// TIA Portal V20 export
FUNCTION_BLOCK "FB_What_Was_Read"   // FB7, LAD
{ S7_Optimized_Access := 'TRUE' }
// stored: AutoNumber false, MemoryReserve 100, SetENOAutomatically false
   VAR_INPUT
      Read_Data_In : "SR-X100W_Read_Data";
   END_VAR
   VAR_OUTPUT
      Read_Data_Out : String[136];
      Serial_Number : String[17];
   END_VAR
BEGIN

REGION Network 1
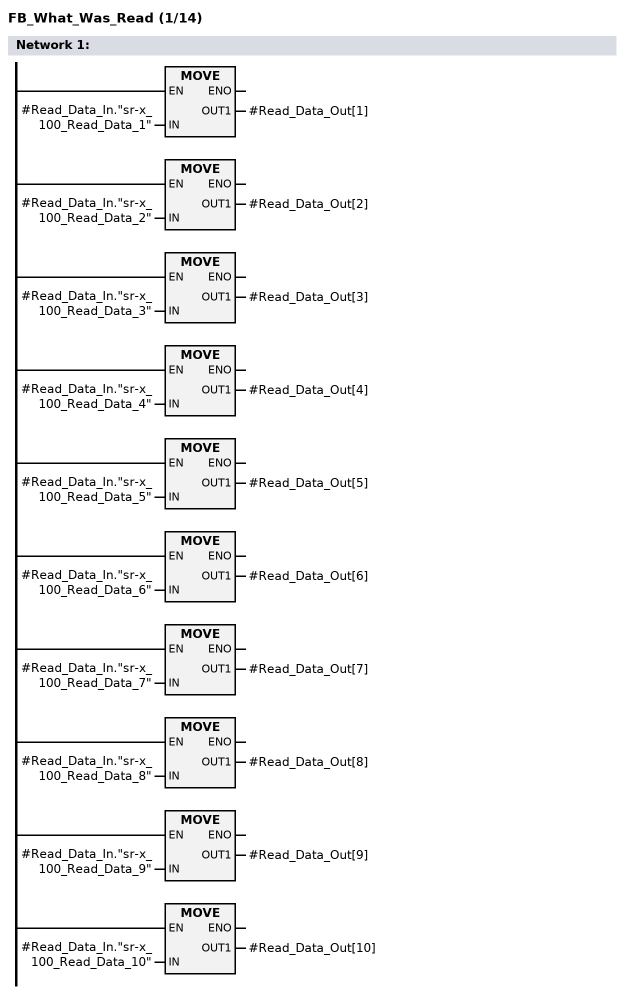
   RUNG wire#powerrail
      Move(in := #Read_Data_In."sr-x_100_Read_Data_1", out1 => #Read_Data_Out[1])
   END_RUNG
   RUNG wire#powerrail
      Move(in := #Read_Data_In."sr-x_100_Read_Data_2", out1 => #Read_Data_Out[2])
   END_RUNG
   RUNG wire#powerrail
      Move(in := #Read_Data_In."sr-x_100_Read_Data_3", out1 => #Read_Data_Out[3])
   END_RUNG
   RUNG wire#powerrail
      Move(in := #Read_Data_In."sr-x_100_Read_Data_4", out1 => #Read_Data_Out[4])
   END_RUNG
   RUNG wire#powerrail
      Move(in := #Read_Data_In."sr-x_100_Read_Data_5", out1 => #Read_Data_Out[5])
   END_RUNG
   RUNG wire#powerrail
      Move(in := #Read_Data_In."sr-x_100_Read_Data_6", out1 => #Read_Data_Out[6])
   END_RUNG
   RUNG wire#powerrail
      Move(in := #Read_Data_In."sr-x_100_Read_Data_7", out1 => #Read_Data_Out[7])
   END_RUNG
   RUNG wire#powerrail
      Move(in := #Read_Data_In."sr-x_100_Read_Data_8", out1 => #Read_Data_Out[8])
   END_RUNG
   RUNG wire#powerrail
      Move(in := #Read_Data_In."sr-x_100_Read_Data_9", out1 => #Read_Data_Out[9])
   END_RUNG
   RUNG wire#powerrail
      Move(in := #Read_Data_In."sr-x_100_Read_Data_10", out1 => #Read_Data_Out[10])
   END_RUNG
   // the same network as SCL:
   #Read_Data_Out[1] := #Read_Data_In."sr-x_100_Read_Data_1";
   #Read_Data_Out[2] := #Read_Data_In."sr-x_100_Read_Data_2";
   #Read_Data_Out[3] := #Read_Data_In."sr-x_100_Read_Data_3";
   #Read_Data_Out[4] := #Read_Data_In."sr-x_100_Read_Data_4";
   #Read_Data_Out[5] := #Read_Data_In."sr-x_100_Read_Data_5";
   #Read_Data_Out[6] := #Read_Data_In."sr-x_100_Read_Data_6";
   #Read_Data_Out[7] := #Read_Data_In."sr-x_100_Read_Data_7";
   #Read_Data_Out[8] := #Read_Data_In."sr-x_100_Read_Data_8";
   #Read_Data_Out[9] := #Read_Data_In."sr-x_100_Read_Data_9";
   #Read_Data_Out[10] := #Read_Data_In."sr-x_100_Read_Data_10";
END_REGION

REGION Network 2
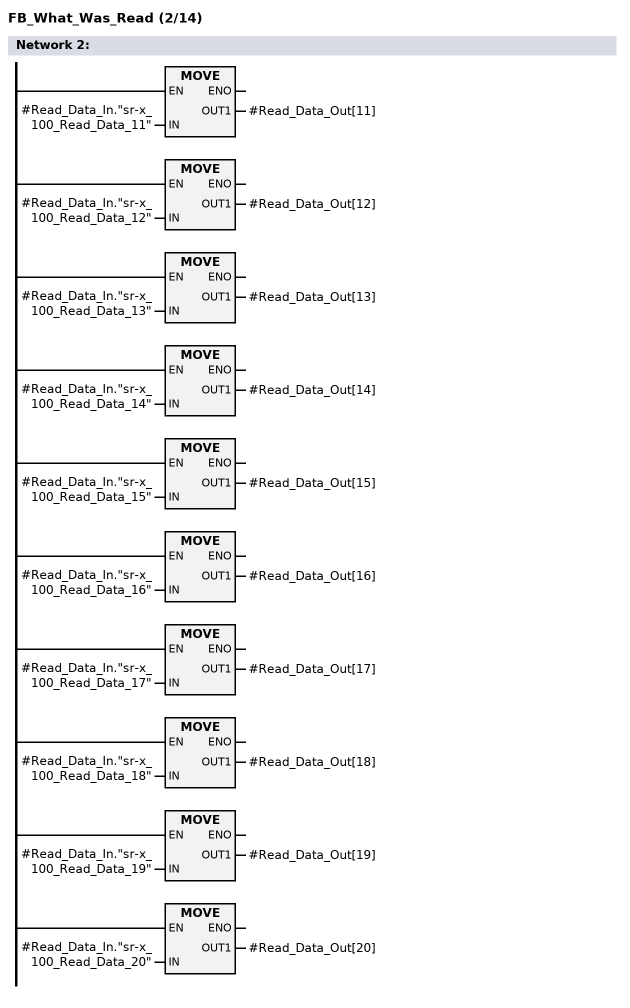
   RUNG wire#powerrail
      Move(in := #Read_Data_In."sr-x_100_Read_Data_11", out1 => #Read_Data_Out[11])
   END_RUNG
   RUNG wire#powerrail
      Move(in := #Read_Data_In."sr-x_100_Read_Data_12", out1 => #Read_Data_Out[12])
   END_RUNG
   RUNG wire#powerrail
      Move(in := #Read_Data_In."sr-x_100_Read_Data_13", out1 => #Read_Data_Out[13])
   END_RUNG
   RUNG wire#powerrail
      Move(in := #Read_Data_In."sr-x_100_Read_Data_14", out1 => #Read_Data_Out[14])
   END_RUNG
   RUNG wire#powerrail
      Move(in := #Read_Data_In."sr-x_100_Read_Data_15", out1 => #Read_Data_Out[15])
   END_RUNG
   RUNG wire#powerrail
      Move(in := #Read_Data_In."sr-x_100_Read_Data_16", out1 => #Read_Data_Out[16])
   END_RUNG
   RUNG wire#powerrail
      Move(in := #Read_Data_In."sr-x_100_Read_Data_17", out1 => #Read_Data_Out[17])
   END_RUNG
   RUNG wire#powerrail
      Move(in := #Read_Data_In."sr-x_100_Read_Data_18", out1 => #Read_Data_Out[18])
   END_RUNG
   RUNG wire#powerrail
      Move(in := #Read_Data_In."sr-x_100_Read_Data_19", out1 => #Read_Data_Out[19])
   END_RUNG
   RUNG wire#powerrail
      Move(in := #Read_Data_In."sr-x_100_Read_Data_20", out1 => #Read_Data_Out[20])
   END_RUNG
   // the same network as SCL:
   #Read_Data_Out[11] := #Read_Data_In."sr-x_100_Read_Data_11";
   #Read_Data_Out[12] := #Read_Data_In."sr-x_100_Read_Data_12";
   #Read_Data_Out[13] := #Read_Data_In."sr-x_100_Read_Data_13";
   #Read_Data_Out[14] := #Read_Data_In."sr-x_100_Read_Data_14";
   #Read_Data_Out[15] := #Read_Data_In."sr-x_100_Read_Data_15";
   #Read_Data_Out[16] := #Read_Data_In."sr-x_100_Read_Data_16";
   #Read_Data_Out[17] := #Read_Data_In."sr-x_100_Read_Data_17";
   #Read_Data_Out[18] := #Read_Data_In."sr-x_100_Read_Data_18";
   #Read_Data_Out[19] := #Read_Data_In."sr-x_100_Read_Data_19";
   #Read_Data_Out[20] := #Read_Data_In."sr-x_100_Read_Data_20";
END_REGION

REGION Network 3
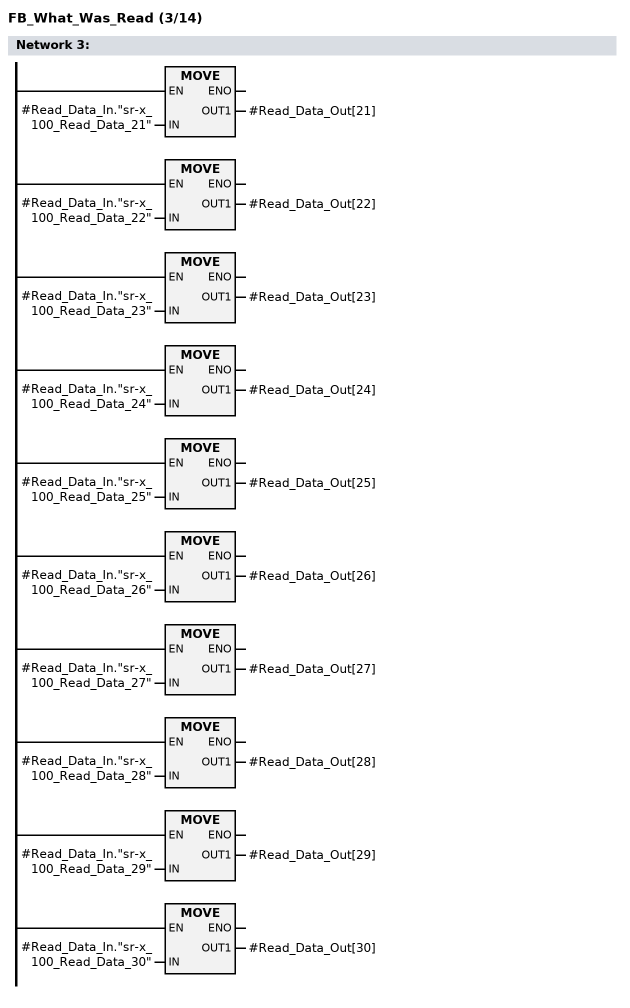
   RUNG wire#powerrail
      Move(in := #Read_Data_In."sr-x_100_Read_Data_21", out1 => #Read_Data_Out[21])
   END_RUNG
   RUNG wire#powerrail
      Move(in := #Read_Data_In."sr-x_100_Read_Data_22", out1 => #Read_Data_Out[22])
   END_RUNG
   RUNG wire#powerrail
      Move(in := #Read_Data_In."sr-x_100_Read_Data_23", out1 => #Read_Data_Out[23])
   END_RUNG
   RUNG wire#powerrail
      Move(in := #Read_Data_In."sr-x_100_Read_Data_24", out1 => #Read_Data_Out[24])
   END_RUNG
   RUNG wire#powerrail
      Move(in := #Read_Data_In."sr-x_100_Read_Data_25", out1 => #Read_Data_Out[25])
   END_RUNG
   RUNG wire#powerrail
      Move(in := #Read_Data_In."sr-x_100_Read_Data_26", out1 => #Read_Data_Out[26])
   END_RUNG
   RUNG wire#powerrail
      Move(in := #Read_Data_In."sr-x_100_Read_Data_27", out1 => #Read_Data_Out[27])
   END_RUNG
   RUNG wire#powerrail
      Move(in := #Read_Data_In."sr-x_100_Read_Data_28", out1 => #Read_Data_Out[28])
   END_RUNG
   RUNG wire#powerrail
      Move(in := #Read_Data_In."sr-x_100_Read_Data_29", out1 => #Read_Data_Out[29])
   END_RUNG
   RUNG wire#powerrail
      Move(in := #Read_Data_In."sr-x_100_Read_Data_30", out1 => #Read_Data_Out[30])
   END_RUNG
   // the same network as SCL:
   #Read_Data_Out[21] := #Read_Data_In."sr-x_100_Read_Data_21";
   #Read_Data_Out[22] := #Read_Data_In."sr-x_100_Read_Data_22";
   #Read_Data_Out[23] := #Read_Data_In."sr-x_100_Read_Data_23";
   #Read_Data_Out[24] := #Read_Data_In."sr-x_100_Read_Data_24";
   #Read_Data_Out[25] := #Read_Data_In."sr-x_100_Read_Data_25";
   #Read_Data_Out[26] := #Read_Data_In."sr-x_100_Read_Data_26";
   #Read_Data_Out[27] := #Read_Data_In."sr-x_100_Read_Data_27";
   #Read_Data_Out[28] := #Read_Data_In."sr-x_100_Read_Data_28";
   #Read_Data_Out[29] := #Read_Data_In."sr-x_100_Read_Data_29";
   #Read_Data_Out[30] := #Read_Data_In."sr-x_100_Read_Data_30";
END_REGION

REGION Network 4
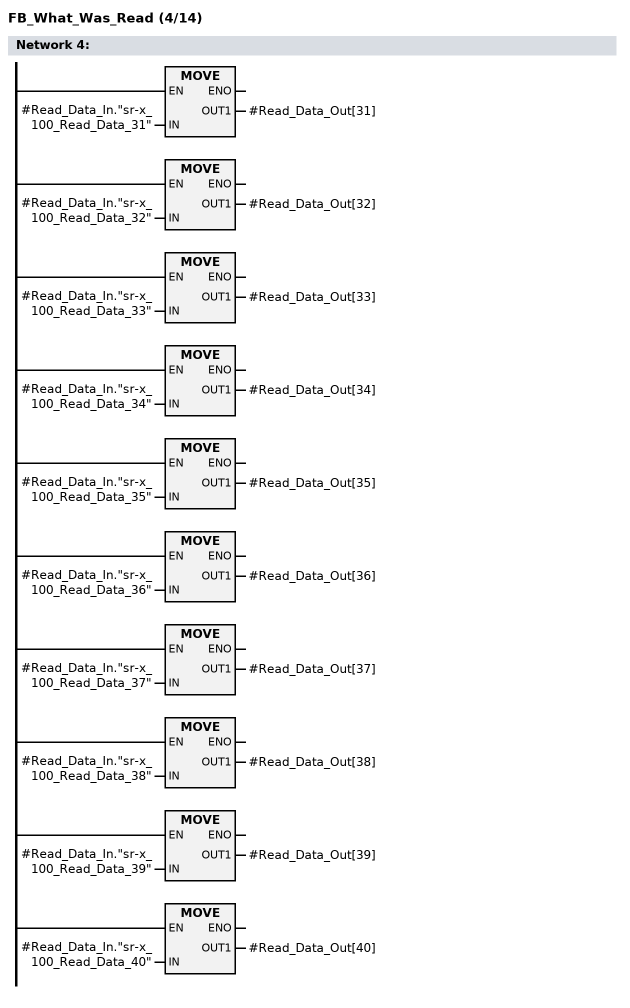
   RUNG wire#powerrail
      Move(in := #Read_Data_In."sr-x_100_Read_Data_31", out1 => #Read_Data_Out[31])
   END_RUNG
   RUNG wire#powerrail
      Move(in := #Read_Data_In."sr-x_100_Read_Data_32", out1 => #Read_Data_Out[32])
   END_RUNG
   RUNG wire#powerrail
      Move(in := #Read_Data_In."sr-x_100_Read_Data_33", out1 => #Read_Data_Out[33])
   END_RUNG
   RUNG wire#powerrail
      Move(in := #Read_Data_In."sr-x_100_Read_Data_34", out1 => #Read_Data_Out[34])
   END_RUNG
   RUNG wire#powerrail
      Move(in := #Read_Data_In."sr-x_100_Read_Data_35", out1 => #Read_Data_Out[35])
   END_RUNG
   RUNG wire#powerrail
      Move(in := #Read_Data_In."sr-x_100_Read_Data_36", out1 => #Read_Data_Out[36])
   END_RUNG
   RUNG wire#powerrail
      Move(in := #Read_Data_In."sr-x_100_Read_Data_37", out1 => #Read_Data_Out[37])
   END_RUNG
   RUNG wire#powerrail
      Move(in := #Read_Data_In."sr-x_100_Read_Data_38", out1 => #Read_Data_Out[38])
   END_RUNG
   RUNG wire#powerrail
      Move(in := #Read_Data_In."sr-x_100_Read_Data_39", out1 => #Read_Data_Out[39])
   END_RUNG
   RUNG wire#powerrail
      Move(in := #Read_Data_In."sr-x_100_Read_Data_40", out1 => #Read_Data_Out[40])
   END_RUNG
   // the same network as SCL:
   #Read_Data_Out[31] := #Read_Data_In."sr-x_100_Read_Data_31";
   #Read_Data_Out[32] := #Read_Data_In."sr-x_100_Read_Data_32";
   #Read_Data_Out[33] := #Read_Data_In."sr-x_100_Read_Data_33";
   #Read_Data_Out[34] := #Read_Data_In."sr-x_100_Read_Data_34";
   #Read_Data_Out[35] := #Read_Data_In."sr-x_100_Read_Data_35";
   #Read_Data_Out[36] := #Read_Data_In."sr-x_100_Read_Data_36";
   #Read_Data_Out[37] := #Read_Data_In."sr-x_100_Read_Data_37";
   #Read_Data_Out[38] := #Read_Data_In."sr-x_100_Read_Data_38";
   #Read_Data_Out[39] := #Read_Data_In."sr-x_100_Read_Data_39";
   #Read_Data_Out[40] := #Read_Data_In."sr-x_100_Read_Data_40";
END_REGION

REGION Network 5
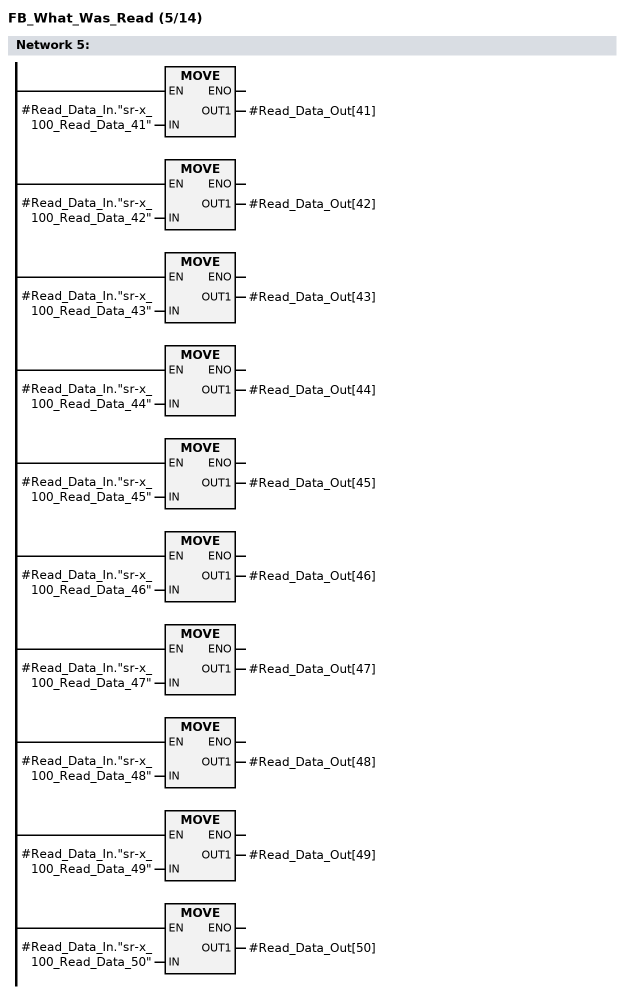
   RUNG wire#powerrail
      Move(in := #Read_Data_In."sr-x_100_Read_Data_41", out1 => #Read_Data_Out[41])
   END_RUNG
   RUNG wire#powerrail
      Move(in := #Read_Data_In."sr-x_100_Read_Data_42", out1 => #Read_Data_Out[42])
   END_RUNG
   RUNG wire#powerrail
      Move(in := #Read_Data_In."sr-x_100_Read_Data_43", out1 => #Read_Data_Out[43])
   END_RUNG
   RUNG wire#powerrail
      Move(in := #Read_Data_In."sr-x_100_Read_Data_44", out1 => #Read_Data_Out[44])
   END_RUNG
   RUNG wire#powerrail
      Move(in := #Read_Data_In."sr-x_100_Read_Data_45", out1 => #Read_Data_Out[45])
   END_RUNG
   RUNG wire#powerrail
      Move(in := #Read_Data_In."sr-x_100_Read_Data_46", out1 => #Read_Data_Out[46])
   END_RUNG
   RUNG wire#powerrail
      Move(in := #Read_Data_In."sr-x_100_Read_Data_47", out1 => #Read_Data_Out[47])
   END_RUNG
   RUNG wire#powerrail
      Move(in := #Read_Data_In."sr-x_100_Read_Data_48", out1 => #Read_Data_Out[48])
   END_RUNG
   RUNG wire#powerrail
      Move(in := #Read_Data_In."sr-x_100_Read_Data_49", out1 => #Read_Data_Out[49])
   END_RUNG
   RUNG wire#powerrail
      Move(in := #Read_Data_In."sr-x_100_Read_Data_50", out1 => #Read_Data_Out[50])
   END_RUNG
   // the same network as SCL:
   #Read_Data_Out[41] := #Read_Data_In."sr-x_100_Read_Data_41";
   #Read_Data_Out[42] := #Read_Data_In."sr-x_100_Read_Data_42";
   #Read_Data_Out[43] := #Read_Data_In."sr-x_100_Read_Data_43";
   #Read_Data_Out[44] := #Read_Data_In."sr-x_100_Read_Data_44";
   #Read_Data_Out[45] := #Read_Data_In."sr-x_100_Read_Data_45";
   #Read_Data_Out[46] := #Read_Data_In."sr-x_100_Read_Data_46";
   #Read_Data_Out[47] := #Read_Data_In."sr-x_100_Read_Data_47";
   #Read_Data_Out[48] := #Read_Data_In."sr-x_100_Read_Data_48";
   #Read_Data_Out[49] := #Read_Data_In."sr-x_100_Read_Data_49";
   #Read_Data_Out[50] := #Read_Data_In."sr-x_100_Read_Data_50";
END_REGION

REGION Network 6
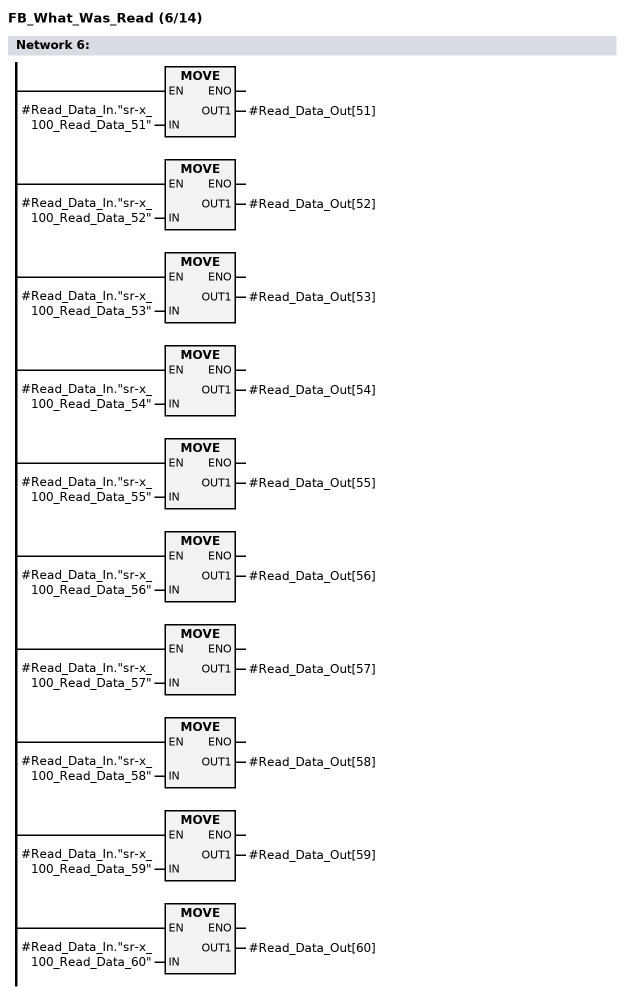
   RUNG wire#powerrail
      Move(in := #Read_Data_In."sr-x_100_Read_Data_51", out1 => #Read_Data_Out[51])
   END_RUNG
   RUNG wire#powerrail
      Move(in := #Read_Data_In."sr-x_100_Read_Data_52", out1 => #Read_Data_Out[52])
   END_RUNG
   RUNG wire#powerrail
      Move(in := #Read_Data_In."sr-x_100_Read_Data_53", out1 => #Read_Data_Out[53])
   END_RUNG
   RUNG wire#powerrail
      Move(in := #Read_Data_In."sr-x_100_Read_Data_54", out1 => #Read_Data_Out[54])
   END_RUNG
   RUNG wire#powerrail
      Move(in := #Read_Data_In."sr-x_100_Read_Data_55", out1 => #Read_Data_Out[55])
   END_RUNG
   RUNG wire#powerrail
      Move(in := #Read_Data_In."sr-x_100_Read_Data_56", out1 => #Read_Data_Out[56])
   END_RUNG
   RUNG wire#powerrail
      Move(in := #Read_Data_In."sr-x_100_Read_Data_57", out1 => #Read_Data_Out[57])
   END_RUNG
   RUNG wire#powerrail
      Move(in := #Read_Data_In."sr-x_100_Read_Data_58", out1 => #Read_Data_Out[58])
   END_RUNG
   RUNG wire#powerrail
      Move(in := #Read_Data_In."sr-x_100_Read_Data_59", out1 => #Read_Data_Out[59])
   END_RUNG
   RUNG wire#powerrail
      Move(in := #Read_Data_In."sr-x_100_Read_Data_60", out1 => #Read_Data_Out[60])
   END_RUNG
   // the same network as SCL:
   #Read_Data_Out[51] := #Read_Data_In."sr-x_100_Read_Data_51";
   #Read_Data_Out[52] := #Read_Data_In."sr-x_100_Read_Data_52";
   #Read_Data_Out[53] := #Read_Data_In."sr-x_100_Read_Data_53";
   #Read_Data_Out[54] := #Read_Data_In."sr-x_100_Read_Data_54";
   #Read_Data_Out[55] := #Read_Data_In."sr-x_100_Read_Data_55";
   #Read_Data_Out[56] := #Read_Data_In."sr-x_100_Read_Data_56";
   #Read_Data_Out[57] := #Read_Data_In."sr-x_100_Read_Data_57";
   #Read_Data_Out[58] := #Read_Data_In."sr-x_100_Read_Data_58";
   #Read_Data_Out[59] := #Read_Data_In."sr-x_100_Read_Data_59";
   #Read_Data_Out[60] := #Read_Data_In."sr-x_100_Read_Data_60";
END_REGION

REGION Network 7
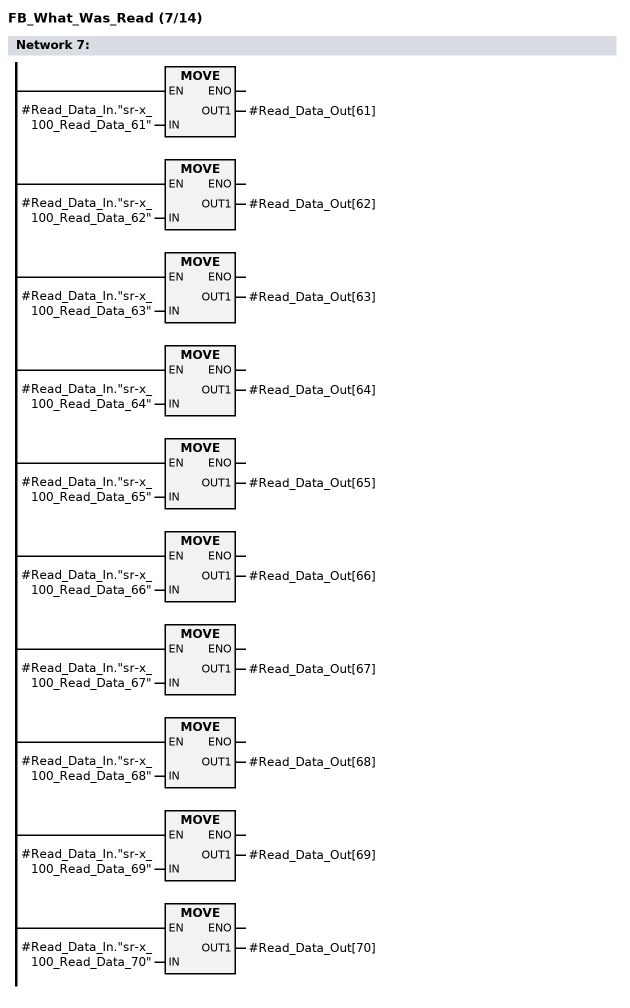
   RUNG wire#powerrail
      Move(in := #Read_Data_In."sr-x_100_Read_Data_61", out1 => #Read_Data_Out[61])
   END_RUNG
   RUNG wire#powerrail
      Move(in := #Read_Data_In."sr-x_100_Read_Data_62", out1 => #Read_Data_Out[62])
   END_RUNG
   RUNG wire#powerrail
      Move(in := #Read_Data_In."sr-x_100_Read_Data_63", out1 => #Read_Data_Out[63])
   END_RUNG
   RUNG wire#powerrail
      Move(in := #Read_Data_In."sr-x_100_Read_Data_64", out1 => #Read_Data_Out[64])
   END_RUNG
   RUNG wire#powerrail
      Move(in := #Read_Data_In."sr-x_100_Read_Data_65", out1 => #Read_Data_Out[65])
   END_RUNG
   RUNG wire#powerrail
      Move(in := #Read_Data_In."sr-x_100_Read_Data_66", out1 => #Read_Data_Out[66])
   END_RUNG
   RUNG wire#powerrail
      Move(in := #Read_Data_In."sr-x_100_Read_Data_67", out1 => #Read_Data_Out[67])
   END_RUNG
   RUNG wire#powerrail
      Move(in := #Read_Data_In."sr-x_100_Read_Data_68", out1 => #Read_Data_Out[68])
   END_RUNG
   RUNG wire#powerrail
      Move(in := #Read_Data_In."sr-x_100_Read_Data_69", out1 => #Read_Data_Out[69])
   END_RUNG
   RUNG wire#powerrail
      Move(in := #Read_Data_In."sr-x_100_Read_Data_70", out1 => #Read_Data_Out[70])
   END_RUNG
   // the same network as SCL:
   #Read_Data_Out[61] := #Read_Data_In."sr-x_100_Read_Data_61";
   #Read_Data_Out[62] := #Read_Data_In."sr-x_100_Read_Data_62";
   #Read_Data_Out[63] := #Read_Data_In."sr-x_100_Read_Data_63";
   #Read_Data_Out[64] := #Read_Data_In."sr-x_100_Read_Data_64";
   #Read_Data_Out[65] := #Read_Data_In."sr-x_100_Read_Data_65";
   #Read_Data_Out[66] := #Read_Data_In."sr-x_100_Read_Data_66";
   #Read_Data_Out[67] := #Read_Data_In."sr-x_100_Read_Data_67";
   #Read_Data_Out[68] := #Read_Data_In."sr-x_100_Read_Data_68";
   #Read_Data_Out[69] := #Read_Data_In."sr-x_100_Read_Data_69";
   #Read_Data_Out[70] := #Read_Data_In."sr-x_100_Read_Data_70";
END_REGION

REGION Network 8
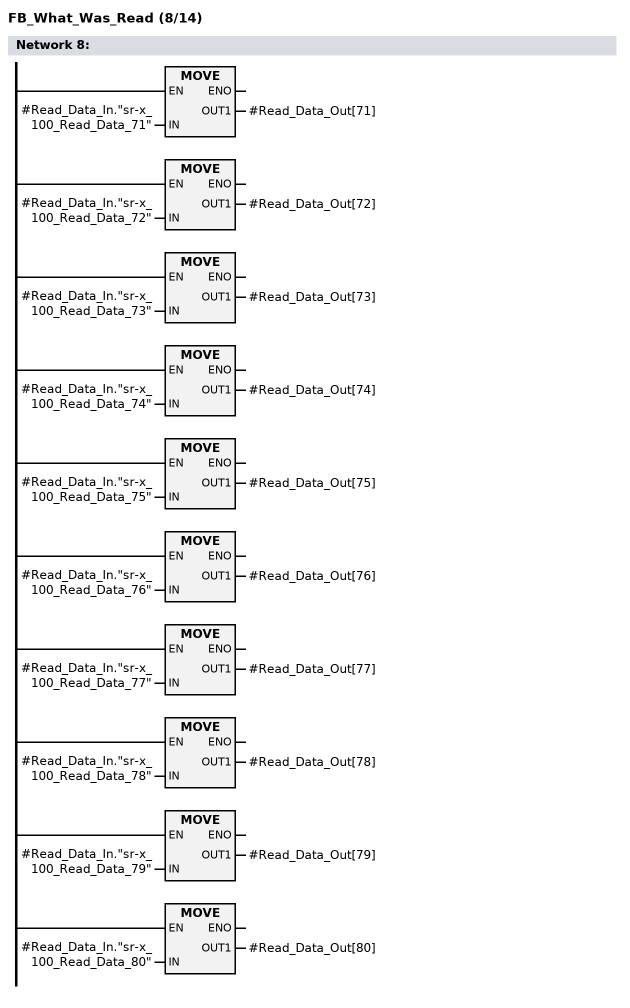
   RUNG wire#powerrail
      Move(in := #Read_Data_In."sr-x_100_Read_Data_71", out1 => #Read_Data_Out[71])
   END_RUNG
   RUNG wire#powerrail
      Move(in := #Read_Data_In."sr-x_100_Read_Data_72", out1 => #Read_Data_Out[72])
   END_RUNG
   RUNG wire#powerrail
      Move(in := #Read_Data_In."sr-x_100_Read_Data_73", out1 => #Read_Data_Out[73])
   END_RUNG
   RUNG wire#powerrail
      Move(in := #Read_Data_In."sr-x_100_Read_Data_74", out1 => #Read_Data_Out[74])
   END_RUNG
   RUNG wire#powerrail
      Move(in := #Read_Data_In."sr-x_100_Read_Data_75", out1 => #Read_Data_Out[75])
   END_RUNG
   RUNG wire#powerrail
      Move(in := #Read_Data_In."sr-x_100_Read_Data_76", out1 => #Read_Data_Out[76])
   END_RUNG
   RUNG wire#powerrail
      Move(in := #Read_Data_In."sr-x_100_Read_Data_77", out1 => #Read_Data_Out[77])
   END_RUNG
   RUNG wire#powerrail
      Move(in := #Read_Data_In."sr-x_100_Read_Data_78", out1 => #Read_Data_Out[78])
   END_RUNG
   RUNG wire#powerrail
      Move(in := #Read_Data_In."sr-x_100_Read_Data_79", out1 => #Read_Data_Out[79])
   END_RUNG
   RUNG wire#powerrail
      Move(in := #Read_Data_In."sr-x_100_Read_Data_80", out1 => #Read_Data_Out[80])
   END_RUNG
   // the same network as SCL:
   #Read_Data_Out[71] := #Read_Data_In."sr-x_100_Read_Data_71";
   #Read_Data_Out[72] := #Read_Data_In."sr-x_100_Read_Data_72";
   #Read_Data_Out[73] := #Read_Data_In."sr-x_100_Read_Data_73";
   #Read_Data_Out[74] := #Read_Data_In."sr-x_100_Read_Data_74";
   #Read_Data_Out[75] := #Read_Data_In."sr-x_100_Read_Data_75";
   #Read_Data_Out[76] := #Read_Data_In."sr-x_100_Read_Data_76";
   #Read_Data_Out[77] := #Read_Data_In."sr-x_100_Read_Data_77";
   #Read_Data_Out[78] := #Read_Data_In."sr-x_100_Read_Data_78";
   #Read_Data_Out[79] := #Read_Data_In."sr-x_100_Read_Data_79";
   #Read_Data_Out[80] := #Read_Data_In."sr-x_100_Read_Data_80";
END_REGION

REGION Network 9
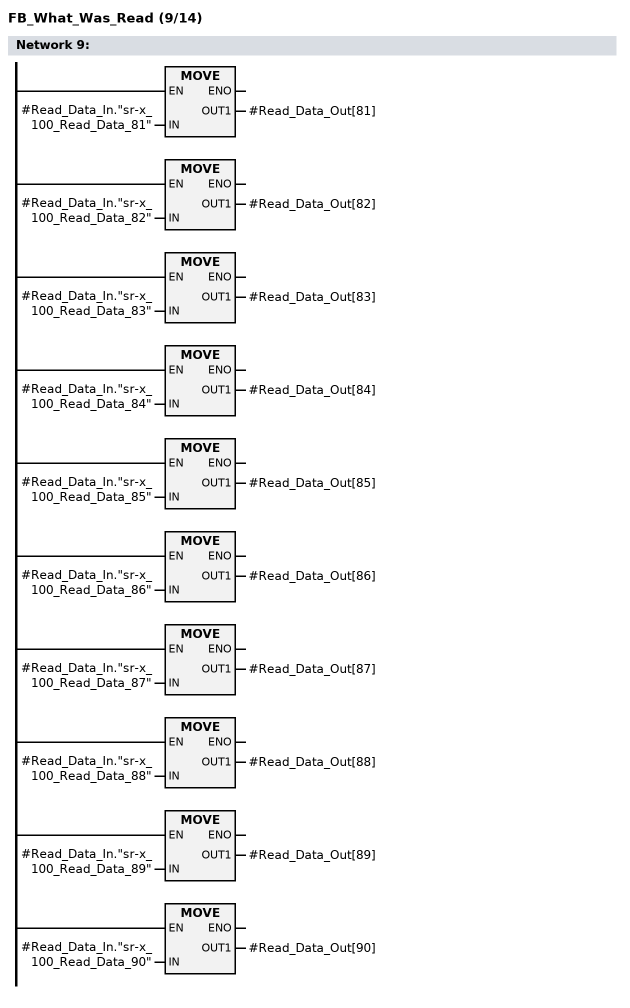
   RUNG wire#powerrail
      Move(in := #Read_Data_In."sr-x_100_Read_Data_81", out1 => #Read_Data_Out[81])
   END_RUNG
   RUNG wire#powerrail
      Move(in := #Read_Data_In."sr-x_100_Read_Data_82", out1 => #Read_Data_Out[82])
   END_RUNG
   RUNG wire#powerrail
      Move(in := #Read_Data_In."sr-x_100_Read_Data_83", out1 => #Read_Data_Out[83])
   END_RUNG
   RUNG wire#powerrail
      Move(in := #Read_Data_In."sr-x_100_Read_Data_84", out1 => #Read_Data_Out[84])
   END_RUNG
   RUNG wire#powerrail
      Move(in := #Read_Data_In."sr-x_100_Read_Data_85", out1 => #Read_Data_Out[85])
   END_RUNG
   RUNG wire#powerrail
      Move(in := #Read_Data_In."sr-x_100_Read_Data_86", out1 => #Read_Data_Out[86])
   END_RUNG
   RUNG wire#powerrail
      Move(in := #Read_Data_In."sr-x_100_Read_Data_87", out1 => #Read_Data_Out[87])
   END_RUNG
   RUNG wire#powerrail
      Move(in := #Read_Data_In."sr-x_100_Read_Data_88", out1 => #Read_Data_Out[88])
   END_RUNG
   RUNG wire#powerrail
      Move(in := #Read_Data_In."sr-x_100_Read_Data_89", out1 => #Read_Data_Out[89])
   END_RUNG
   RUNG wire#powerrail
      Move(in := #Read_Data_In."sr-x_100_Read_Data_90", out1 => #Read_Data_Out[90])
   END_RUNG
   // the same network as SCL:
   #Read_Data_Out[81] := #Read_Data_In."sr-x_100_Read_Data_81";
   #Read_Data_Out[82] := #Read_Data_In."sr-x_100_Read_Data_82";
   #Read_Data_Out[83] := #Read_Data_In."sr-x_100_Read_Data_83";
   #Read_Data_Out[84] := #Read_Data_In."sr-x_100_Read_Data_84";
   #Read_Data_Out[85] := #Read_Data_In."sr-x_100_Read_Data_85";
   #Read_Data_Out[86] := #Read_Data_In."sr-x_100_Read_Data_86";
   #Read_Data_Out[87] := #Read_Data_In."sr-x_100_Read_Data_87";
   #Read_Data_Out[88] := #Read_Data_In."sr-x_100_Read_Data_88";
   #Read_Data_Out[89] := #Read_Data_In."sr-x_100_Read_Data_89";
   #Read_Data_Out[90] := #Read_Data_In."sr-x_100_Read_Data_90";
END_REGION

REGION Network 10
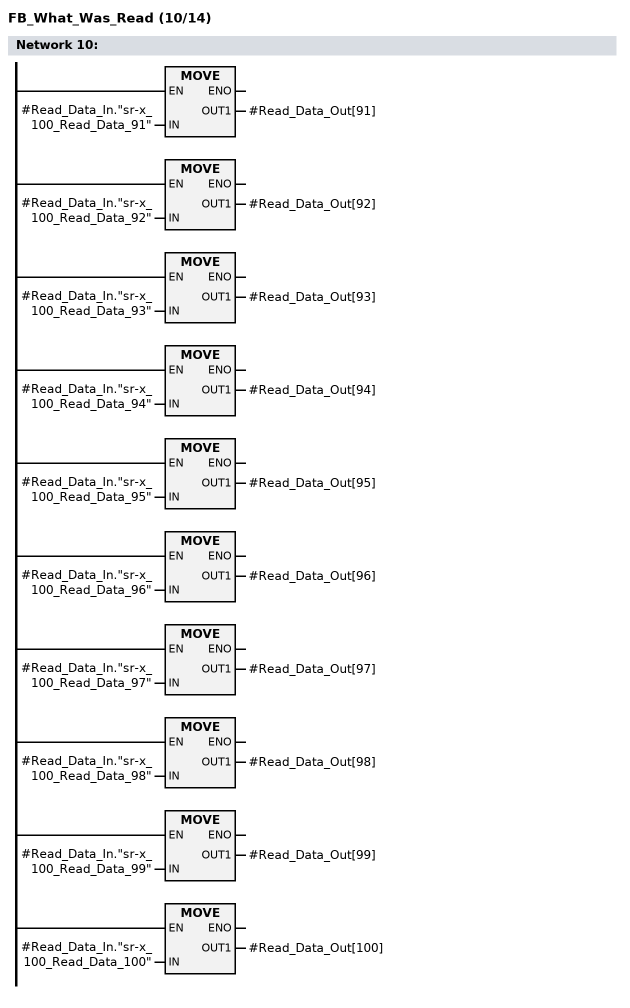
   RUNG wire#powerrail
      Move(in := #Read_Data_In."sr-x_100_Read_Data_91", out1 => #Read_Data_Out[91])
   END_RUNG
   RUNG wire#powerrail
      Move(in := #Read_Data_In."sr-x_100_Read_Data_92", out1 => #Read_Data_Out[92])
   END_RUNG
   RUNG wire#powerrail
      Move(in := #Read_Data_In."sr-x_100_Read_Data_93", out1 => #Read_Data_Out[93])
   END_RUNG
   RUNG wire#powerrail
      Move(in := #Read_Data_In."sr-x_100_Read_Data_94", out1 => #Read_Data_Out[94])
   END_RUNG
   RUNG wire#powerrail
      Move(in := #Read_Data_In."sr-x_100_Read_Data_95", out1 => #Read_Data_Out[95])
   END_RUNG
   RUNG wire#powerrail
      Move(in := #Read_Data_In."sr-x_100_Read_Data_96", out1 => #Read_Data_Out[96])
   END_RUNG
   RUNG wire#powerrail
      Move(in := #Read_Data_In."sr-x_100_Read_Data_97", out1 => #Read_Data_Out[97])
   END_RUNG
   RUNG wire#powerrail
      Move(in := #Read_Data_In."sr-x_100_Read_Data_98", out1 => #Read_Data_Out[98])
   END_RUNG
   RUNG wire#powerrail
      Move(in := #Read_Data_In."sr-x_100_Read_Data_99", out1 => #Read_Data_Out[99])
   END_RUNG
   RUNG wire#powerrail
      Move(in := #Read_Data_In."sr-x_100_Read_Data_100", out1 => #Read_Data_Out[100])
   END_RUNG
   // the same network as SCL:
   #Read_Data_Out[91] := #Read_Data_In."sr-x_100_Read_Data_91";
   #Read_Data_Out[92] := #Read_Data_In."sr-x_100_Read_Data_92";
   #Read_Data_Out[93] := #Read_Data_In."sr-x_100_Read_Data_93";
   #Read_Data_Out[94] := #Read_Data_In."sr-x_100_Read_Data_94";
   #Read_Data_Out[95] := #Read_Data_In."sr-x_100_Read_Data_95";
   #Read_Data_Out[96] := #Read_Data_In."sr-x_100_Read_Data_96";
   #Read_Data_Out[97] := #Read_Data_In."sr-x_100_Read_Data_97";
   #Read_Data_Out[98] := #Read_Data_In."sr-x_100_Read_Data_98";
   #Read_Data_Out[99] := #Read_Data_In."sr-x_100_Read_Data_99";
   #Read_Data_Out[100] := #Read_Data_In."sr-x_100_Read_Data_100";
END_REGION

REGION Network 11
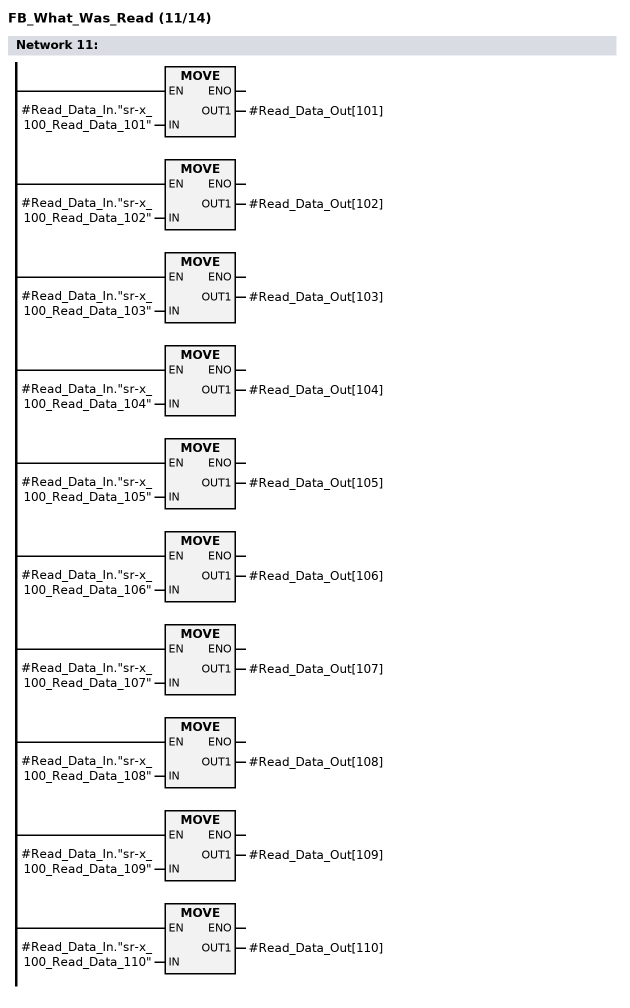
   RUNG wire#powerrail
      Move(in := #Read_Data_In."sr-x_100_Read_Data_101", out1 => #Read_Data_Out[101])
   END_RUNG
   RUNG wire#powerrail
      Move(in := #Read_Data_In."sr-x_100_Read_Data_102", out1 => #Read_Data_Out[102])
   END_RUNG
   RUNG wire#powerrail
      Move(in := #Read_Data_In."sr-x_100_Read_Data_103", out1 => #Read_Data_Out[103])
   END_RUNG
   RUNG wire#powerrail
      Move(in := #Read_Data_In."sr-x_100_Read_Data_104", out1 => #Read_Data_Out[104])
   END_RUNG
   RUNG wire#powerrail
      Move(in := #Read_Data_In."sr-x_100_Read_Data_105", out1 => #Read_Data_Out[105])
   END_RUNG
   RUNG wire#powerrail
      Move(in := #Read_Data_In."sr-x_100_Read_Data_106", out1 => #Read_Data_Out[106])
   END_RUNG
   RUNG wire#powerrail
      Move(in := #Read_Data_In."sr-x_100_Read_Data_107", out1 => #Read_Data_Out[107])
   END_RUNG
   RUNG wire#powerrail
      Move(in := #Read_Data_In."sr-x_100_Read_Data_108", out1 => #Read_Data_Out[108])
   END_RUNG
   RUNG wire#powerrail
      Move(in := #Read_Data_In."sr-x_100_Read_Data_109", out1 => #Read_Data_Out[109])
   END_RUNG
   RUNG wire#powerrail
      Move(in := #Read_Data_In."sr-x_100_Read_Data_110", out1 => #Read_Data_Out[110])
   END_RUNG
   // the same network as SCL:
   #Read_Data_Out[101] := #Read_Data_In."sr-x_100_Read_Data_101";
   #Read_Data_Out[102] := #Read_Data_In."sr-x_100_Read_Data_102";
   #Read_Data_Out[103] := #Read_Data_In."sr-x_100_Read_Data_103";
   #Read_Data_Out[104] := #Read_Data_In."sr-x_100_Read_Data_104";
   #Read_Data_Out[105] := #Read_Data_In."sr-x_100_Read_Data_105";
   #Read_Data_Out[106] := #Read_Data_In."sr-x_100_Read_Data_106";
   #Read_Data_Out[107] := #Read_Data_In."sr-x_100_Read_Data_107";
   #Read_Data_Out[108] := #Read_Data_In."sr-x_100_Read_Data_108";
   #Read_Data_Out[109] := #Read_Data_In."sr-x_100_Read_Data_109";
   #Read_Data_Out[110] := #Read_Data_In."sr-x_100_Read_Data_110";
END_REGION

REGION Network 12
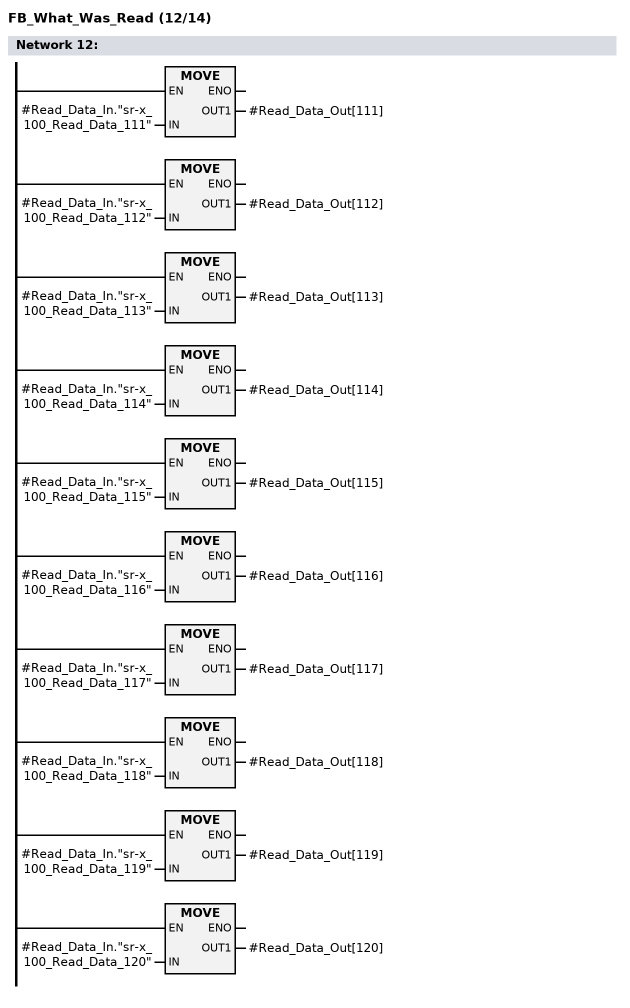
   RUNG wire#powerrail
      Move(in := #Read_Data_In."sr-x_100_Read_Data_111", out1 => #Read_Data_Out[111])
   END_RUNG
   RUNG wire#powerrail
      Move(in := #Read_Data_In."sr-x_100_Read_Data_112", out1 => #Read_Data_Out[112])
   END_RUNG
   RUNG wire#powerrail
      Move(in := #Read_Data_In."sr-x_100_Read_Data_113", out1 => #Read_Data_Out[113])
   END_RUNG
   RUNG wire#powerrail
      Move(in := #Read_Data_In."sr-x_100_Read_Data_114", out1 => #Read_Data_Out[114])
   END_RUNG
   RUNG wire#powerrail
      Move(in := #Read_Data_In."sr-x_100_Read_Data_115", out1 => #Read_Data_Out[115])
   END_RUNG
   RUNG wire#powerrail
      Move(in := #Read_Data_In."sr-x_100_Read_Data_116", out1 => #Read_Data_Out[116])
   END_RUNG
   RUNG wire#powerrail
      Move(in := #Read_Data_In."sr-x_100_Read_Data_117", out1 => #Read_Data_Out[117])
   END_RUNG
   RUNG wire#powerrail
      Move(in := #Read_Data_In."sr-x_100_Read_Data_118", out1 => #Read_Data_Out[118])
   END_RUNG
   RUNG wire#powerrail
      Move(in := #Read_Data_In."sr-x_100_Read_Data_119", out1 => #Read_Data_Out[119])
   END_RUNG
   RUNG wire#powerrail
      Move(in := #Read_Data_In."sr-x_100_Read_Data_120", out1 => #Read_Data_Out[120])
   END_RUNG
   // the same network as SCL:
   #Read_Data_Out[111] := #Read_Data_In."sr-x_100_Read_Data_111";
   #Read_Data_Out[112] := #Read_Data_In."sr-x_100_Read_Data_112";
   #Read_Data_Out[113] := #Read_Data_In."sr-x_100_Read_Data_113";
   #Read_Data_Out[114] := #Read_Data_In."sr-x_100_Read_Data_114";
   #Read_Data_Out[115] := #Read_Data_In."sr-x_100_Read_Data_115";
   #Read_Data_Out[116] := #Read_Data_In."sr-x_100_Read_Data_116";
   #Read_Data_Out[117] := #Read_Data_In."sr-x_100_Read_Data_117";
   #Read_Data_Out[118] := #Read_Data_In."sr-x_100_Read_Data_118";
   #Read_Data_Out[119] := #Read_Data_In."sr-x_100_Read_Data_119";
   #Read_Data_Out[120] := #Read_Data_In."sr-x_100_Read_Data_120";
END_REGION

REGION Network 13
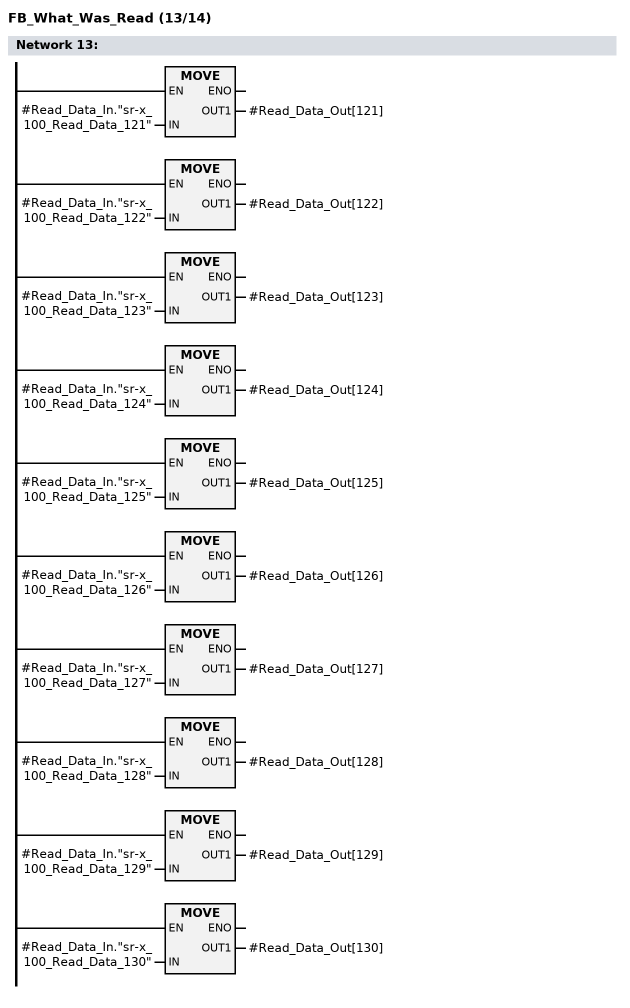
   RUNG wire#powerrail
      Move(in := #Read_Data_In."sr-x_100_Read_Data_121", out1 => #Read_Data_Out[121])
   END_RUNG
   RUNG wire#powerrail
      Move(in := #Read_Data_In."sr-x_100_Read_Data_122", out1 => #Read_Data_Out[122])
   END_RUNG
   RUNG wire#powerrail
      Move(in := #Read_Data_In."sr-x_100_Read_Data_123", out1 => #Read_Data_Out[123])
   END_RUNG
   RUNG wire#powerrail
      Move(in := #Read_Data_In."sr-x_100_Read_Data_124", out1 => #Read_Data_Out[124])
   END_RUNG
   RUNG wire#powerrail
      Move(in := #Read_Data_In."sr-x_100_Read_Data_125", out1 => #Read_Data_Out[125])
   END_RUNG
   RUNG wire#powerrail
      Move(in := #Read_Data_In."sr-x_100_Read_Data_126", out1 => #Read_Data_Out[126])
   END_RUNG
   RUNG wire#powerrail
      Move(in := #Read_Data_In."sr-x_100_Read_Data_127", out1 => #Read_Data_Out[127])
   END_RUNG
   RUNG wire#powerrail
      Move(in := #Read_Data_In."sr-x_100_Read_Data_128", out1 => #Read_Data_Out[128])
   END_RUNG
   RUNG wire#powerrail
      Move(in := #Read_Data_In."sr-x_100_Read_Data_129", out1 => #Read_Data_Out[129])
   END_RUNG
   RUNG wire#powerrail
      Move(in := #Read_Data_In."sr-x_100_Read_Data_130", out1 => #Read_Data_Out[130])
   END_RUNG
   // the same network as SCL:
   #Read_Data_Out[121] := #Read_Data_In."sr-x_100_Read_Data_121";
   #Read_Data_Out[122] := #Read_Data_In."sr-x_100_Read_Data_122";
   #Read_Data_Out[123] := #Read_Data_In."sr-x_100_Read_Data_123";
   #Read_Data_Out[124] := #Read_Data_In."sr-x_100_Read_Data_124";
   #Read_Data_Out[125] := #Read_Data_In."sr-x_100_Read_Data_125";
   #Read_Data_Out[126] := #Read_Data_In."sr-x_100_Read_Data_126";
   #Read_Data_Out[127] := #Read_Data_In."sr-x_100_Read_Data_127";
   #Read_Data_Out[128] := #Read_Data_In."sr-x_100_Read_Data_128";
   #Read_Data_Out[129] := #Read_Data_In."sr-x_100_Read_Data_129";
   #Read_Data_Out[130] := #Read_Data_In."sr-x_100_Read_Data_130";
END_REGION

REGION Network 14
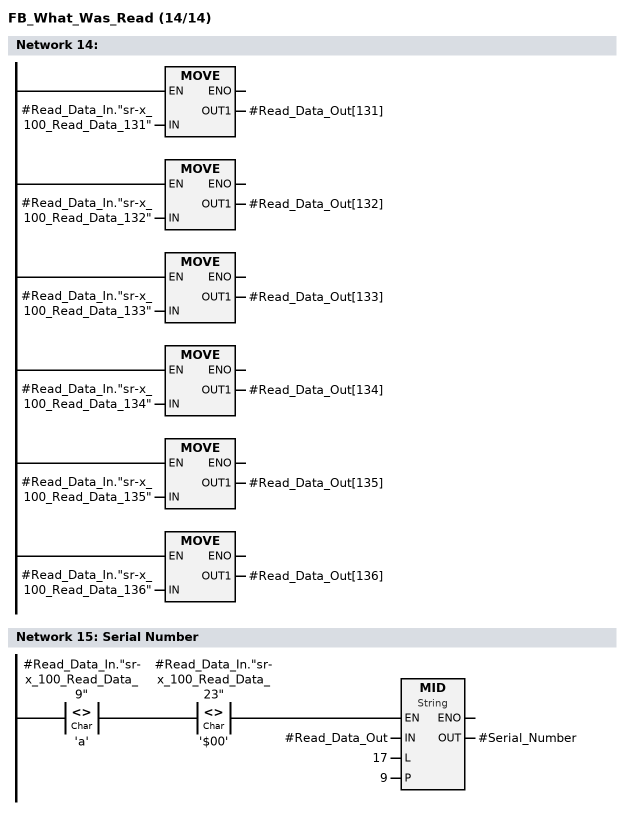
   RUNG wire#powerrail
      Move(in := #Read_Data_In."sr-x_100_Read_Data_131", out1 => #Read_Data_Out[131])
   END_RUNG
   RUNG wire#powerrail
      Move(in := #Read_Data_In."sr-x_100_Read_Data_132", out1 => #Read_Data_Out[132])
   END_RUNG
   RUNG wire#powerrail
      Move(in := #Read_Data_In."sr-x_100_Read_Data_133", out1 => #Read_Data_Out[133])
   END_RUNG
   RUNG wire#powerrail
      Move(in := #Read_Data_In."sr-x_100_Read_Data_134", out1 => #Read_Data_Out[134])
   END_RUNG
   RUNG wire#powerrail
      Move(in := #Read_Data_In."sr-x_100_Read_Data_135", out1 => #Read_Data_Out[135])
   END_RUNG
   RUNG wire#powerrail
      Move(in := #Read_Data_In."sr-x_100_Read_Data_136", out1 => #Read_Data_Out[136])
   END_RUNG
   // the same network as SCL:
   #Read_Data_Out[131] := #Read_Data_In."sr-x_100_Read_Data_131";
   #Read_Data_Out[132] := #Read_Data_In."sr-x_100_Read_Data_132";
   #Read_Data_Out[133] := #Read_Data_In."sr-x_100_Read_Data_133";
   #Read_Data_Out[134] := #Read_Data_In."sr-x_100_Read_Data_134";
   #Read_Data_Out[135] := #Read_Data_In."sr-x_100_Read_Data_135";
   #Read_Data_Out[136] := #Read_Data_In."sr-x_100_Read_Data_136";
END_REGION

REGION Network 15: Serial Number
   RUNG wire#powerrail
      { S7_Templates := "SrcType := Char" } NE_Contact(in1 := #Read_Data_In."sr-x_100_Read_Data_9", in2 := 'a')
      { S7_Templates := "SrcType := Char" } NE_Contact(in1 := #Read_Data_In."sr-x_100_Read_Data_23", in2 := '$00')
      { S7_Templates := "value_type := String" } MID(IN := #Read_Data_Out, L := 17, P := 9, OUT => #Serial_Number)
   END_RUNG
   // the same network as SCL:
   IF (#Read_Data_In."sr-x_100_Read_Data_9" <> 'a') AND (#Read_Data_In."sr-x_100_Read_Data_23" <> '$00') THEN
       MID(IN := #Read_Data_Out, L := 17, P := 9, OUT => #Serial_Number);
   END_IF;
END_REGION
END_FUNCTION_BLOCK
